FUNCTION F_HighestInt : INT
VAR_INPUT
	Value1																: INT;
	Value2																: INT;
END_VAR
VAR
END_VAR

// F_Highest2
// Rev 1.0 - March 14, 2024

F_HighestInt																:= SEL(Value1 > Value2, Value2, Value1);

END_FUNCTION

(* stored: Version 1.1.0.1, ProductVersion 3.1.4024.12
   POU F_HighestInt: Id {1eefb2dd-a801-40ca-83f4-983ff054a5e4}, SpecialFunc None *)
